REGION Network 42: Status signals
   // ▀▀▀▀▀▀▀▀▀▀▀▀▀▀▀▀▀▀▀▀▀▀▀▀▀▀▀▀▀▀▀▀▀▀▀▀▀▀▀▀▀▀▀▀
   // The status signals for faults, alarms and warnings are either duplicates of the message signals 
   // (signals beginning with msg_) or logical combinations of them.
   // 
   // The following is a full list of the status signals:
   // 
   //  UT31001_Dy_DevValveIsol (full contents)
   //  ――――――――――――――――――――――――――――――――――――――――――
   //  SIGNAL NAME          FUNCTION                     TYPE
   //  ――――――――――――――――――――――――――――――――――――――――――
   //  status_Operating        STATUS — Valve is changing state           Bool
   //                      (1 = changing state, 0 = fixed state)
   //  status_Fault            STATUS — Valve is in fault              Bool
   //                      (1 = fault present, 0 = healthy)
   //  status_Energised        STATUS — Valve output is on              Bool
   //                      (1 = energised, 0 = deenergised)
   //  status_Aut           STATUS — Automatic mode active           Bool
   //                      (1 = auto mode on, 0 = auto mode off)
   //  status_Man          STATUS — Manual mode active             Bool
   //                      (1 = man mode on, 0 = man mode off)
   //  status_EStop          STATUS — E_STOP safety signal is active         Bool
   //                      (1 = active, 0 = healthy)
   //  status_Trip        STATUS — TRIP signal is active             Bool
   //                      (1 = active, 0 = healthy)
   //  status_Ilock         STATUS — INTERLOCK signal is active            Bool
   //                      (1 = active, 0 = healthy)
   //  status_Perm        STATUS — PERMISSIVE signal is active           Bool
   //                      (1 = active, 0 = healthy)
   //  status_BypassOn        STATUS — Valve is in bypass mode          Bool
   //                      (1 = Simulation mode, 0 = normal)
   //  status_SimOn           STATUS — Valve is in simulation mode               Bool
   //                      (1 = Simulation mode, 0 = normal)
   //  status_RemoteOn       STATUS — Valve is in remote mode                  Bool
   //                      (1 = Remote mode, 0 = normal)
   //  status_LocalOn         STATUS — Valve is in local mode                    Bool
   //                      (1 = Local mode, 0 = normal)
   //  status_RLOff         STATUS — Valve is in ALL mode                   Bool
   //                      (1 = ALL mode, 0 = normal)
   //  ――――――――――――――――――――――――――――――――――――――――――
   // ▄▄▄▄▄▄▄▄▄▄▄▄▄▄▄▄▄▄▄▄▄▄▄▄▄▄▄▄▄▄▄▄▄▄▄▄▄▄▄▄▄▄▄▄
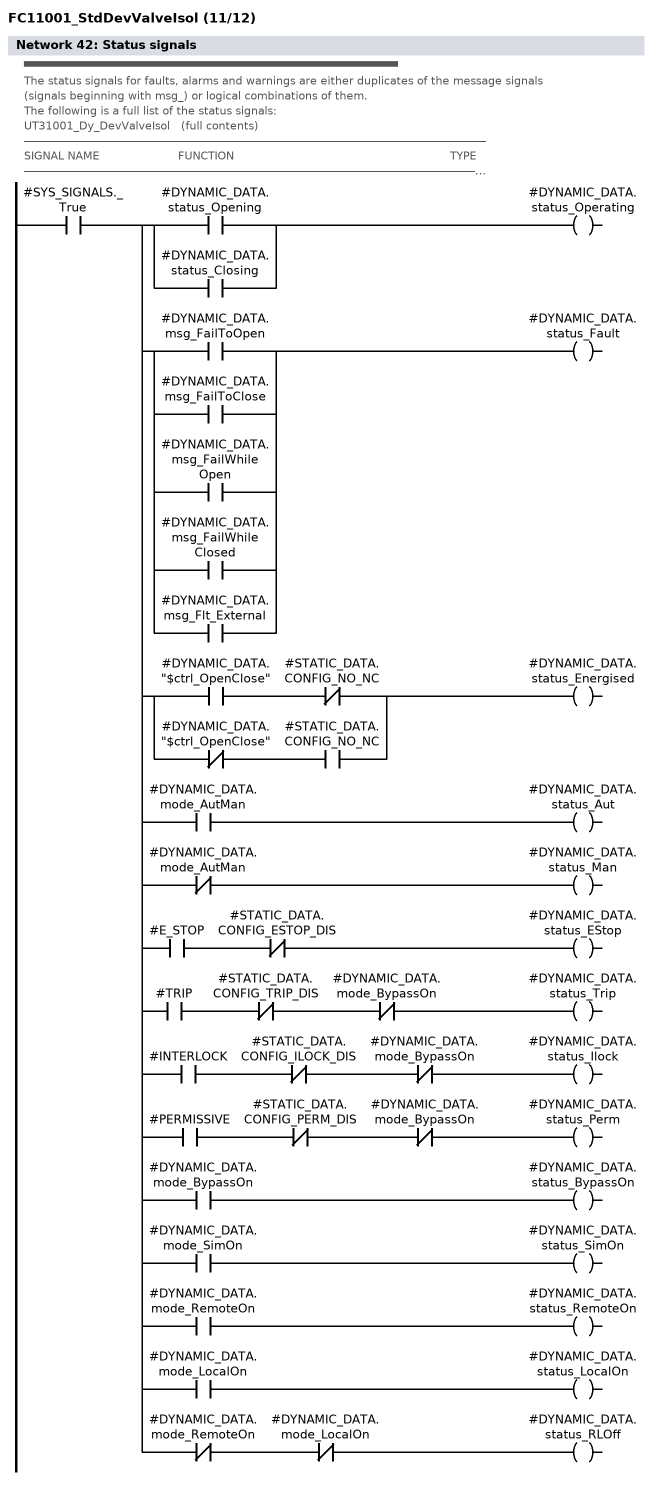
   RUNG wire#powerrail
      Contact( #SYS_SIGNALS._True )
      wire#w1
      Contact( #DYNAMIC_DATA.status_Opening )
      wire#w2
      Coil( #DYNAMIC_DATA.status_Operating )
   END_RUNG
   RUNG wire#w1
      Contact( #DYNAMIC_DATA.status_Closing )
   END_RUNG wire#w2
   RUNG wire#w1
      Contact( #DYNAMIC_DATA.msg_FailToOpen )
      wire#w3
      Coil( #DYNAMIC_DATA.status_Fault )
   END_RUNG
   RUNG wire#w1
      Contact( #DYNAMIC_DATA.msg_FailToClose )
   END_RUNG wire#w3
   RUNG wire#w1
      Contact( #DYNAMIC_DATA.msg_FailWhileOpen )
   END_RUNG wire#w3
   RUNG wire#w1
      Contact( #DYNAMIC_DATA.msg_FailWhileClosed )
   END_RUNG wire#w3
   RUNG wire#w1
      Contact( #DYNAMIC_DATA.msg_Flt_External )
   END_RUNG wire#w3
   RUNG wire#w1
      Contact( #DYNAMIC_DATA."$ctrl_OpenClose" )
      I_Contact( #STATIC_DATA.CONFIG_NO_NC )
      wire#w4
      Coil( #DYNAMIC_DATA.status_Energised )
   END_RUNG
   RUNG wire#w1
      I_Contact( #DYNAMIC_DATA."$ctrl_OpenClose" )
      Contact( #STATIC_DATA.CONFIG_NO_NC )
   END_RUNG wire#w4
   RUNG wire#w1
      Contact( #DYNAMIC_DATA.mode_AutMan )
      Coil( #DYNAMIC_DATA.status_Aut )
   END_RUNG
   RUNG wire#w1
      I_Contact( #DYNAMIC_DATA.mode_AutMan )
      Coil( #DYNAMIC_DATA.status_Man )
   END_RUNG
   RUNG wire#w1
      Contact( #E_STOP )
      I_Contact( #STATIC_DATA.CONFIG_ESTOP_DIS )
      Coil( #DYNAMIC_DATA.status_EStop )
   END_RUNG
   RUNG wire#w1
      Contact( #TRIP )
      I_Contact( #STATIC_DATA.CONFIG_TRIP_DIS )
      I_Contact( #DYNAMIC_DATA.mode_BypassOn )
      Coil( #DYNAMIC_DATA.status_Trip )
   END_RUNG
   RUNG wire#w1
      Contact( #INTERLOCK )
      I_Contact( #STATIC_DATA.CONFIG_ILOCK_DIS )
      I_Contact( #DYNAMIC_DATA.mode_BypassOn )
      Coil( #DYNAMIC_DATA.status_Ilock )
   END_RUNG
   RUNG wire#w1
      Contact( #PERMISSIVE )
      I_Contact( #STATIC_DATA.CONFIG_PERM_DIS )
      I_Contact( #DYNAMIC_DATA.mode_BypassOn )
      Coil( #DYNAMIC_DATA.status_Perm )
   END_RUNG
   RUNG wire#w1
      Contact( #DYNAMIC_DATA.mode_BypassOn )
      Coil( #DYNAMIC_DATA.status_BypassOn )
   END_RUNG
   RUNG wire#w1
      Contact( #DYNAMIC_DATA.mode_SimOn )
      Coil( #DYNAMIC_DATA.status_SimOn )
   END_RUNG
   RUNG wire#w1
      Contact( #DYNAMIC_DATA.mode_RemoteOn )
      Coil( #DYNAMIC_DATA.status_RemoteOn )
   END_RUNG
   RUNG wire#w1
      Contact( #DYNAMIC_DATA.mode_LocalOn )
      Coil( #DYNAMIC_DATA.status_LocalOn )
   END_RUNG
   RUNG wire#w1
      I_Contact( #DYNAMIC_DATA.mode_RemoteOn )
      I_Contact( #DYNAMIC_DATA.mode_LocalOn )
      Coil( #DYNAMIC_DATA.status_RLOff )
   END_RUNG
   // the same network as SCL:
   #DYNAMIC_DATA.status_Operating := #SYS_SIGNALS._True AND (#DYNAMIC_DATA.status_Opening OR #DYNAMIC_DATA.status_Closing);
   #DYNAMIC_DATA.status_Fault := #SYS_SIGNALS._True AND (#DYNAMIC_DATA.msg_FailToOpen OR #DYNAMIC_DATA.msg_FailToClose OR #DYNAMIC_DATA.msg_FailWhileOpen OR #DYNAMIC_DATA.msg_FailWhileClosed OR #DYNAMIC_DATA.msg_Flt_External);
   #DYNAMIC_DATA.status_Energised := #SYS_SIGNALS._True AND ((#DYNAMIC_DATA."$ctrl_OpenClose" AND NOT #STATIC_DATA.CONFIG_NO_NC) OR (NOT #DYNAMIC_DATA."$ctrl_OpenClose" AND #STATIC_DATA.CONFIG_NO_NC));
   #DYNAMIC_DATA.status_Aut := #SYS_SIGNALS._True AND #DYNAMIC_DATA.mode_AutMan;
   #DYNAMIC_DATA.status_Man := #SYS_SIGNALS._True AND NOT #DYNAMIC_DATA.mode_AutMan;
   #DYNAMIC_DATA.status_EStop := #SYS_SIGNALS._True AND #E_STOP AND NOT #STATIC_DATA.CONFIG_ESTOP_DIS;
   #DYNAMIC_DATA.status_Trip := #SYS_SIGNALS._True AND #TRIP AND NOT #STATIC_DATA.CONFIG_TRIP_DIS AND NOT #DYNAMIC_DATA.mode_BypassOn;
   #DYNAMIC_DATA.status_Ilock := #SYS_SIGNALS._True AND #INTERLOCK AND NOT #STATIC_DATA.CONFIG_ILOCK_DIS AND NOT #DYNAMIC_DATA.mode_BypassOn;
   #DYNAMIC_DATA.status_Perm := #SYS_SIGNALS._True AND #PERMISSIVE AND NOT #STATIC_DATA.CONFIG_PERM_DIS AND NOT #DYNAMIC_DATA.mode_BypassOn;
   #DYNAMIC_DATA.status_BypassOn := #SYS_SIGNALS._True AND #DYNAMIC_DATA.mode_BypassOn;
   #DYNAMIC_DATA.status_SimOn := #SYS_SIGNALS._True AND #DYNAMIC_DATA.mode_SimOn;
   #DYNAMIC_DATA.status_RemoteOn := #SYS_SIGNALS._True AND #DYNAMIC_DATA.mode_RemoteOn;
   #DYNAMIC_DATA.status_LocalOn := #SYS_SIGNALS._True AND #DYNAMIC_DATA.mode_LocalOn;
   #DYNAMIC_DATA.status_RLOff := #SYS_SIGNALS._True AND NOT #DYNAMIC_DATA.mode_RemoteOn AND NOT #DYNAMIC_DATA.mode_LocalOn;
END_REGION

REGION Network 43: Output driver
   // ▀▀▀▀▀▀▀▀▀▀▀▀▀▀▀▀▀▀▀▀▀▀▀▀▀▀▀▀▀▀▀▀▀▀▀▀▀▀▀▀▀▀▀▀
   // Copy the required energised/deenergised state (status_Energised) to the valve output 
   // parameter (#OPERATE)
   // ▄▄▄▄▄▄▄▄▄▄▄▄▄▄▄▄▄▄▄▄▄▄▄▄▄▄▄▄▄▄▄▄▄▄▄▄▄▄▄▄▄▄▄▄
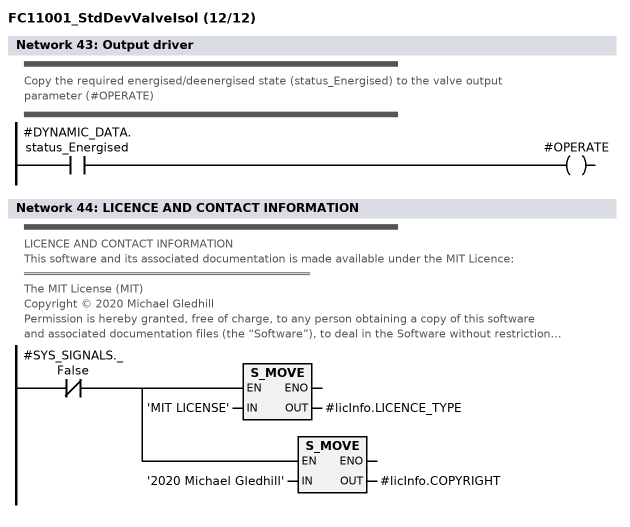
   RUNG wire#powerrail
      Contact( #DYNAMIC_DATA.status_Energised )
      Coil( #OPERATE )
   END_RUNG
   // the same network as SCL:
   #OPERATE := #DYNAMIC_DATA.status_Energised;
END_REGION

REGION Network 44: LICENCE AND CONTACT INFORMATION
   // ▀▀▀▀▀▀▀▀▀▀▀▀▀▀▀▀▀▀▀▀▀▀▀▀▀▀▀▀▀▀▀▀▀▀▀▀▀▀▀▀▀▀▀▀
   // LICENCE AND CONTACT INFORMATION
   // 
   // This software and its associated documentation is made available under the MIT Licence:
   // 
   // ════════════════════════════════════════════
   // 
   // The MIT License (MIT)
   // 
   // Copyright © 2020 Michael Gledhill
   // 
   // Permission is hereby granted, free of charge, to any person obtaining a copy of this software 
   // and associated documentation files (the “Software”), to deal in the Software without restriction, 
   // including without limitation the rights to use, copy, modify, merge, publish, distribute, 
   // sublicense, and/or sell copies of the Software, and to permit persons to whom the Software is 
   // furnished to do so, subject to the following conditions: 
   // 
   // The above copyright notice and this permission notice shall be included in all copies or 
   // substantial portions of the Software.
   // 
   // THE SOFTWARE IS PROVIDED “AS IS”, WITHOUT WARRANTY OF ANY KIND, EXPRESS OR IMPLIED, 
   // INCLUDING BUT NOT LIMITED TO THE WARRANTIES OF MERCHANTABILITY, FITNESS FOR A 
   // PARTICULAR PURPOSE AND NON-INFRINGEMENT. IN NO EVENT SHALL THE AUTHORS OR COPYRIGHT 
   // HOLDERS BE LIABLE FOR ANY CLAIM, DAMAGES OR OTHER LIABILITY, WHETHER IN AN ACTION OF 
   // CONTRACT, TORT OR OTHERWISE, ARISING FROM, OUT OF OR IN CONNECTION WITH THE SOFTWARE 
   // OR THE USE OR OTHER DEALINGS IN THE SOFTWARE.
   // 
   // ════════════════════════════════════════════
   //                    ┌────────────┐
   // You can reach the author by email here:   │  mg@practicalseries.com  │
   //                    └────────────┘
   // Questions, corrections, constructive criticism and complaints (polite ones) are invited.
   RUNG wire#powerrail
      I_Contact( #SYS_SIGNALS._False )
      wire#w1
      S_Move(in := 'MIT LICENSE', out => #licInfo.LICENCE_TYPE)
   END_RUNG
   RUNG wire#w1
      S_Move(in := '2020 Michael Gledhill', out => #licInfo.COPYRIGHT)
   END_RUNG
   // the same network as SCL:
   IF NOT #SYS_SIGNALS._False THEN
       #licInfo.LICENCE_TYPE := 'MIT LICENSE';
       #licInfo.COPYRIGHT := '2020 Michael Gledhill';
   END_IF;
END_REGION
END_FUNCTION
